FUNCTION_BLOCK FB_LedIndicator
VAR_INPUT
	by_brightness				: BYTE; // in %
	io							: ST_LEDstrip_IOvars;
END_VAR

VAR_IN_OUT CONSTANT
	st_params					: st_ledstrip_params;
END_VAR

VAR CONSTANT
	w_ID						: WORD := eObject_ID.Enclosure_LED;
END_VAR

VAR_OUTPUT
	get						: ST_Ledstrip_get;
END_VAR

VAR
	
END_VAR

VAR
	Write						: TON;
	CommFaultOffDelay			: TOF;
	aw_LED_ModbusOutputRegs		: ARRAY [0..10] OF WORD;
	b_enable					: BOOL := TRUE;
	WriteRegs					: FB_MBWriteRegs;
	t_RefreshTime				: TIME := T#1S;
	t_TimeOut					: TIME := T#1S;
END_VAR

SetData();

IF b_enable THEN
	Write(IN:= NOT write.Q, PT := t_RefreshTime);
	CommFaultOffDelay(IN:= writeregs.bError, PT := T#5S, Q => get.b_LedCommFault);
	
	WriteRegs(sIPAddr := st_params.IP,
		nTCPPort := 502,
		nUnitID := 16#FF,
		nQuantity := st_params.noRegisters,
		nMBaddr := 0,
		cbLength := SIZEOF(aw_LED_ModbusOutputRegs),
		pSrcAddr := ADR(aw_LED_ModbusOutputRegs),
		bExecute := Write.Q,
		tTimeOut := t_Timeout);	
END_IF

METHOD PUBLIC GetDiagnostics
VAR_IN_OUT
	AddError		: ARRAY [*] OF FB_AddErrorST;
	a_ActiveEvents	: ARRAY [*] OF ST_ErrorStruct;
	w_Index			: WORD;
END_VAR

VAR_OUTPUT
	b_errorActive	: BOOL;
	b_warningActive	: BOOL;
END_VAR

VAR
	by_errCt	: BYTE;
	by_warnCt	: BYTE;
END_VAR
	(*Led Com fault*)		AddError[w_Index](
		b_ErrorTrig			:= get.b_LedCommFault,
		out_ST_Error			:= a_ActiveEvents[w_Index],
		w_ErrorID					:= 1,
		e_ObjectID				:=  eObject_ID.Enclosure_LED,
		s_Message				:= 'communication fault',
		e_sev					:= eseverity.info,
		b_AutoClear			:= TRUE
		);
		w_Index := w_Index +1;
END_METHOD

METHOD PUBLIC Reset : BOOL

VAR_INST
	ton_ResetPulse			: TON := (pt:=T#500MS);

END_VAR
IF get.b_LedCommFault THEN
	ton_resetPulse(IN:= NOT ton_ResetPulse.Q);
	b_enable := ton_ResetPulse.Q;
ELSE
	b_enable := TRUE;
END_IF

reset := NOT get.b_LedCommFault;
END_METHOD

METHOD PRIVATE SetData


VAR
	by_Status 					: BYTE;
	by_mode						: BYTE := 0;
END_VAR

VAR_INST
	TON_ledstripColorPulse			: TON := (PT:=T#500MS);
	b_toggle						: BOOL;
END_VAR
TON_ledstripColorPulse(IN:= NOT TON_ledstripColorPulse.Q);
IF ton_ledstripColorPulse.Q THEN
	b_toggle := NOT b_toggle;
END_IF


 // Get status (ePu500)
IF io.b_Error THEN
	by_Status := 4;
ELSIF io.b_warning THEN 
	by_Status := 3;
ELSIF io.b_attention THEN 
	by_Status := 2;
ELSIF io.b_Normal THEN   
	by_Status := 1;
ELSE // neutral
	by_status := 0;
END_IF

IF io.r_DCCurrent < -10 THEN
	by_mode := 1; //charging
ELSIF io.r_DCCurrent > 10 THEN
	by_mode := 2; //discharging
ELSE
	by_mode := 0; // idle
END_IF


// Fill in regs
aw_LED_ModbusOutputRegs[0] := TO_WORD(MAX(LIMIT(0,io.r_SOC,100) *2.55,1));   				// Battery usable state of charge (0.1%)
aw_LED_ModbusOutputRegs[1] := TO_WORD(by_Status); // Battery status (0: Neutral, 1: Normal, 2: attention, 3: Warning, 4: Error)
aw_LED_ModbusOutputRegs[2] := TO_WORD(by_mode);	// 0 = idle, 1 = charging, 2 = discharging				
aw_LED_ModbusOutputRegs[3] := TO_WORD(SEL(io.b_off, LIMIT(10, by_brightness, 100), 0) * 2.55); 					// LED strip brightness (0-255)
aw_LED_ModbusOutputRegs[4] := st_params.Numleds; 	
aw_LED_ModbusOutputRegs[5] := 0; 	  
aw_LED_ModbusOutputRegs[6] := st_params.ColorOrder;
END_METHOD

END_FUNCTION_BLOCK

(* stored: Version 1.1.0.1, ProductVersion 3.1.4024.12
   POU FB_LedIndicator: Id {50068ffc-9ab7-4765-9343-61ec41c921a7}, SpecialFunc None
   Method GetDiagnostics: Id {3a536bba-6768-443a-9dbc-eb3b6a8d2df8}
   Method Reset: Id {d067fcd7-4ae1-44bc-9482-a55675def6c7}
   Method SetData: Id {dcd32f3f-2552-4239-915d-3b09790f80db} *)
